GLOBALCONSTANTS isobus (* Global constants *)
  (* Standard: 61499-1 *)
  (* Version 1.0, 2023-10-22, franz *)
  VAR_GLOBAL CONSTANT
    ID_NULL : UINT := UINT#16#FFFF;
  END_VAR
END_GLOBALCONSTANTS
